INTERFACE I_XP_Station EXTENDS I_CH_Object

{attribute 'monitoring':='call'}
//Track on which the station is located
PROPERTY AccocietedTrack : I_XP_Track
GET
END_GET
END_PROPERTY

METHOD AddMoverToQueue : HRESULT
VAR_INPUT
	ipMover : I_XP_Mover;
END_VAR
END_METHOD

{attribute 'monitoring':='call'}
//List of movers managed by this station
PROPERTY AssignedMovers : I_CH_List
GET
END_GET
END_PROPERTY

//Call this Methode whith seq 0->100, and wait each step until S_OK is returned
METHOD Configure : HRESULT
VAR_INPUT
	nSeq : UINT; //0->100
END_VAR
END_METHOD

{attribute 'monitoring':='call'}
PROPERTY CtsEmptySpaceInQueue : UDINT
GET
END_GET
END_PROPERTY

{attribute 'monitoring':='call'}
PROPERTY CtsMoversInQueue : UDINT
GET
END_GET
END_PROPERTY

METHOD DeleteMoversQueue : HRESULT
VAR_INPUT
END_VAR
END_METHOD

{attribute 'monitoring':='call'}
PROPERTY Filter : STRING
GET
END_GET
SET
END_SET
END_PROPERTY

{attribute 'monitoring':='call'}
PROPERTY MoverAccAtExit : MC_LREAL //[mm/s² on Track] Every mover that leaves or passes the station gets this new acceleration as a target.
GET
END_GET
END_PROPERTY

{attribute 'monitoring':='call'}
PROPERTY MoverDecAtExit : MC_LREAL //[mm/s² on Track] Every mover that leaves or passes the station gets this new deceleration as a target.
GET
END_GET
END_PROPERTY

{attribute 'monitoring':='call'}
//[mm] Every mover that leaves or passes the station gets this new gap as a target.
PROPERTY MoverGapAtExit : LREAL
GET
END_GET
SET
END_SET
END_PROPERTY

{attribute 'monitoring':='call'}
PROPERTY MoverQueueSize : UINT
GET
END_GET
END_PROPERTY

{attribute 'monitoring':='call'}
PROPERTY MoversInPlace : BOOL
GET
END_GET
END_PROPERTY

{attribute 'monitoring':='call'}
PROPERTY MoverVelocityAtExit : MC_LREAL //[mm/s on Track] Every mover that leaves or passes the station gets this new velocity as a target.
GET
END_GET
END_PROPERTY

{attribute 'monitoring':='call'}
//List of paths that lead to stations before this station
PROPERTY PathsAhead : I_CH_List
GET
END_GET
END_PROPERTY

{attribute 'monitoring':='call'}
//List of paths that lead to stations behind this station
PROPERTY PathsBehinde : I_CH_List
GET
END_GET
END_PROPERTY

{attribute 'monitoring':='call'}
//[mm] from the beginning of the assigned track
PROPERTY PositionOnTrack : LREAL
GET
END_GET
END_PROPERTY

{attribute 'monitoring':='call'}
//Position on the assigned track
PROPERTY PositionOnTrackXY : REFERENCE TO PositionXY
GET
END_GET
END_PROPERTY

{attribute 'monitoring':='call'}
//Planned position, not necessarily on the track
PROPERTY PositionXY : REFERENCE TO  PositionXY
GET
END_GET
END_PROPERTY

//The movers currently in this station must leave the station. 
//The movers actively search for a destination, but only leave if a new destination is available.
METHOD PushMoversOutOfStation : HRESULT
VAR_INPUT
END_VAR
END_METHOD

{attribute 'monitoring':='call'}
//prevent further movers from entering the station, 
//e.g. to prevent a collision. All movers that are already moving to reach this station will be stopped with a stop 
//and restarted with Ready True.
PROPERTY ReadyToRecvMovers : BOOL
GET
END_GET
END_PROPERTY

METHOD SendMoversToStation : I_CH_Feedback //All movers in the station are sent to this destination
VAR_INPUT
	sTargetStation: STRING;//unique station name or group of stations
END_VAR
END_METHOD

{attribute 'monitoring':='call'}
//List of stations before this station
PROPERTY StationsAhead : I_CH_List
GET
END_GET
END_PROPERTY

{attribute 'monitoring':='call'}
//List of stations behinde this station
PROPERTY StationsBehinde : I_CH_List
GET
END_GET
END_PROPERTY

{attribute 'monitoring':='call'}
PROPERTY TargetGroupe : STRING
GET
END_GET
END_PROPERTY

METHOD Update : HRESULT
VAR_INPUT
END_VAR
END_METHOD

END_INTERFACE

(* stored: Version 1.1.0.1, ProductVersion 3.1.4024.12
   Itf I_XP_Station: Id {3d974a17-7bf1-45ea-a1bb-e6a1207524fe}
   Property AccocietedTrack: Id {f1f8fb4d-f5e8-4293-ab6b-e19a472e59da}
   Get Get: Id {9a483f3b-2b37-4504-9722-e1528e1cf396}
   Method AddMoverToQueue: Id {c4da7942-2d63-4214-a839-5ac13c1f072a}
   Property AssignedMovers: Id {8cd89700-2be3-47cc-925c-cee79fa842fd}
   Get Get: Id {5cb2b908-d7cd-4ce9-b194-f1a72e296d0e}
   Method Configure: Id {bc350bf6-8abf-47b4-bb67-c376b4ee15bf}
   Property CtsEmptySpaceInQueue: Id {1897c6d1-ecca-457a-bc9c-de434b01ee29}
   Get Get: Id {c3c1562f-b9ef-48e7-b8a1-983628ddd9ed}
   Property CtsMoversInQueue: Id {7a8ac52b-d8b4-46c2-af98-ad00f1a720fd}
   Get Get: Id {92717f46-0e8a-4f98-a1ea-f807eabab1a8}
   Method DeleteMoversQueue: Id {4df869e3-43c4-41fb-9494-0537850d74ad}
   Property Filter: Id {b167339c-04a5-499d-b56c-05cfe366bab8}
   Get Get: Id {d27c3f71-e718-48a5-9c99-1fbf8433c1ec}
   Set Set: Id {84bcc4bb-4e27-4145-8bbf-6e51a5e53ce9}
   Property MoverAccAtExit: Id {f6d020e5-5ae6-4fbd-871f-3ced3aa3dc8b}
   Get Get: Id {b5390215-9e0d-4f6c-9007-25100751e160}
   Property MoverDecAtExit: Id {8fa4da0d-915b-49f1-8edc-36b8ff2b8b12}
   Get Get: Id {858d3fd4-dc9e-49c8-bbb9-316153a4983d}
   Property MoverGapAtExit: Id {c5e80f53-5b29-456f-a007-b994ba73eb10}
   Get Get: Id {d12a186c-96cc-44d7-b200-559663ffbefe}
   Set Set: Id {4beb67d3-bee0-4a44-b3b8-42b2d2bb2df6}
   Property MoverQueueSize: Id {80986d81-19b1-42b6-af07-3458ea2c0b50}
   Get Get: Id {a8272dda-c098-47e7-9f23-a03ea55f0d6c}
   Property MoversInPlace: Id {0ac094d8-21dd-4bed-9c5a-66becba2a927}
   Get Get: Id {3f8d5da7-f95f-4c2c-bcd6-5db015e4c0cf}
   Property MoverVelocityAtExit: Id {5d9d42a8-4ac4-4607-a031-f46c9e2704cd}
   Get Get: Id {f3533885-93e6-4be9-9c15-489b563bc262}
   Property PathsAhead: Id {0435d021-9e32-4506-b359-a43a32741a81}
   Get Get: Id {5f01485c-717f-489c-8c8d-6a47f50c4fc7}
   Property PathsBehinde: Id {3794d1c7-4c72-4c97-9a4e-656ae7fc93cb}
   Get Get: Id {60fa4d14-36f0-4e0e-97ef-19447f215401}
   Property PositionOnTrack: Id {1995ed67-50eb-4b29-8b06-4f9329ae5e7c}
   Get Get: Id {3a9d7479-0ed2-4bfb-9888-de466a1001f9}
   Property PositionOnTrackXY: Id {08286a01-cfce-45ac-a931-ea486a69b4f2}
   Get Get: Id {a9dbad2f-8ea7-4f41-a263-b3e5c35b4ffd}
   Property PositionXY: Id {18df1069-0957-468b-96bf-9f0ba52731b7}
   Get Get: Id {09416665-bf5e-4716-be3f-5e44e14b1445}
   Method PushMoversOutOfStation: Id {49ec1e31-cfe0-48bc-8941-6d431ddc0c3b}
   Property ReadyToRecvMovers: Id {587a5dac-08bc-4c6e-ac52-3ddc0f3e20f9}
   Get Get: Id {c6b87ecc-2972-4dc7-aaa9-af4d00ddfb47}
   Method SendMoversToStation: Id {ea1d0745-bc3a-4dc6-9685-a98523a491dd}
   Property StationsAhead: Id {7a9bb62c-e314-49ec-bae2-5edb8a19790b}
   Get Get: Id {64a1eb89-5f81-45dc-a19d-a6cd0bd0ccae}
   Property StationsBehinde: Id {bad569b2-399c-48ff-8fc7-9c3af9c67938}
   Get Get: Id {82d39e6d-dfe2-40d9-b338-aebf2b2841a9}
   Property TargetGroupe: Id {7f0da163-013b-42b5-9a58-a5d05bf925bc}
   Get Get: Id {9d892f15-0aaf-412a-a3d2-c381f6cd5d76}
   Method Update: Id {88efa7a1-495a-495d-b209-6ee84bfa33b0} *)
